{attribute 'linkalways'} 
{attribute 'no_explicit_call' := 'This FB is a CLASS and must be accessed using methods or properties'}
{attribute 'enable_dynamic_creation'}
FUNCTION_BLOCK FINAL MAX_LREAL EXTENDS Node
VAR
	in1 : _LREAL(0.0);
	in2 : _LREAL(0.0);
	out : _LREAL(0.0);
END_VAR

METHOD PUBLIC Clone : I_Node
VAR
	pNode : POINTER TO MAX_LREAL;
END_VAR
pNode := __NEW(MAX_LREAL);
Clone := pNode^;
END_METHOD

METHOD FB_init : BOOL
VAR_INPUT
	bInitRetains : BOOL; // if TRUE, the retain variables are initialized (warm start / cold start)
	bInCopyCode : BOOL;  // if TRUE, the instance afterwards gets moved into the copy code (online change)
END_VAR
AddInput('in1',THIS^.in1);
AddInput('in2',THIS^.in2);
AddOutput('out', THIS^.out);
END_METHOD

METHOD PROTECTED OnExecute
VAR
END_VAR
out.Value := MAX(in1.Value, in2.Value);
END_METHOD

END_FUNCTION_BLOCK

(* stored: Version 1.1.0.1, ProductVersion 3.1.4024.15
   POU MAX_LREAL: Id {892fcdfb-7d23-4b6b-ab41-0600a141c31c}, SpecialFunc None
   Folder Constructor: Id {fb24d8ee-8478-4403-9829-1cb10f5453f5}
   Method Clone: Id {44e6477c-4b78-4bb1-919a-b6ce745e78f2}
   Method FB_init: Id {3eb3b880-f881-4a66-b7be-babf030062ab}
   Method OnExecute: Id {8cd2d6f6-5f6d-425f-9fde-8bd34a82ffb9} *)
